PROGRAM Loaders
VAR
	Loader_1: Loader;
	Loader_2: Loader;
	Loader_3: Loader;
	FB_Loader_1: FB_Loader;
	FB_Loader_2: FB_Loader;
	FB_Loader_3: FB_Loader;
END_VAR

// note: this text did not pass the execution check against the stored diagram
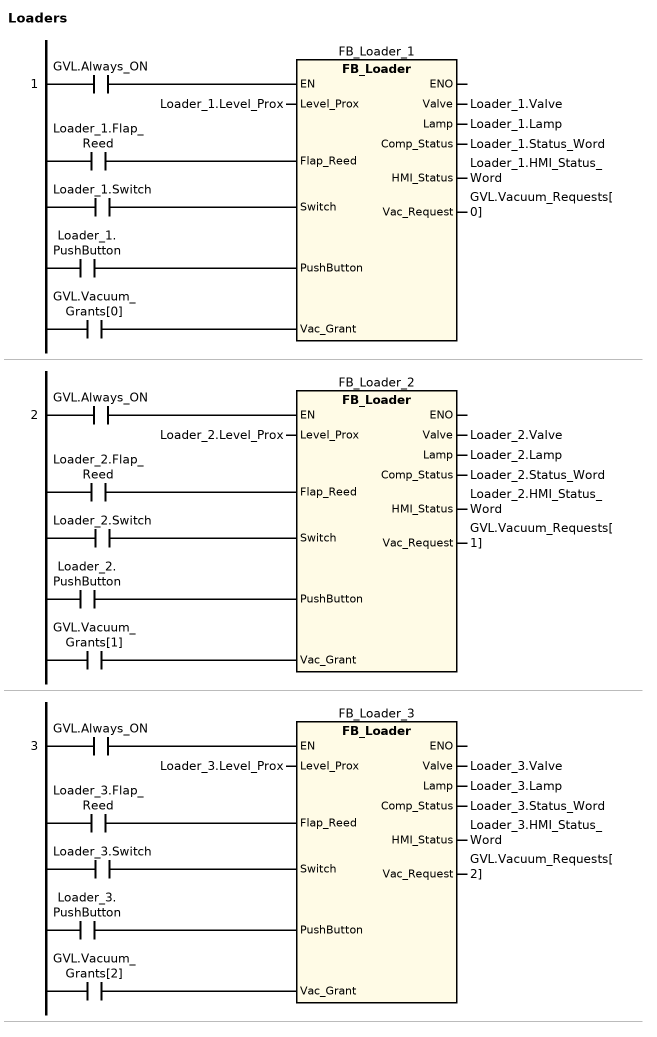
// NETWORK 1
FB_Loader_1(
    EN := GVL.Always_ON,
    Level_Prox := Loader_1.Level_Prox,
    Flap_Reed := Loader_1.Flap_Reed,
    Switch := Loader_1.Switch,
    PushButton := Loader_1.PushButton,
    Vac_Grant := GVL.Vacuum_Grants[0],
    Valve => Loader_1.Valve,
    Lamp => Loader_1.Lamp,
    Comp_Status => Loader_1.Status_Word,
    HMI_Status => Loader_1.HMI_Status_Word,
    Vac_Request => GVL.Vacuum_Requests[0]); // FB_Loader

// NETWORK 2
FB_Loader_2(
    EN := GVL.Always_ON,
    Level_Prox := Loader_2.Level_Prox,
    Flap_Reed := Loader_2.Flap_Reed,
    Switch := Loader_2.Switch,
    PushButton := Loader_2.PushButton,
    Vac_Grant := GVL.Vacuum_Grants[1],
    Valve => Loader_2.Valve,
    Lamp => Loader_2.Lamp,
    Comp_Status => Loader_2.Status_Word,
    HMI_Status => Loader_2.HMI_Status_Word,
    Vac_Request => GVL.Vacuum_Requests[1]); // FB_Loader

// NETWORK 3
FB_Loader_3(
    EN := GVL.Always_ON,
    Level_Prox := Loader_3.Level_Prox,
    Flap_Reed := Loader_3.Flap_Reed,
    Switch := Loader_3.Switch,
    PushButton := Loader_3.PushButton,
    Vac_Grant := GVL.Vacuum_Grants[2],
    Valve => Loader_3.Valve,
    Lamp => Loader_3.Lamp,
    Comp_Status => Loader_3.Status_Word,
    HMI_Status => Loader_3.HMI_Status_Word,
    Vac_Request => GVL.Vacuum_Requests[2]); // FB_Loader

END_PROGRAM

(* stored: Version 1.1.0.1, ProductVersion 3.1.4024.13
   POU Loaders: Id {dac9b70e-e2e1-4da2-bbd2-5d9b244dd886}, SpecialFunc None *)
